PROGRAM Motion_Step_ST
VAR
    Vision_OK_Trig     : R_TRIG;             // 비전 OK 상승엣지(결과 캡처)
    VisionQueue        : FB_VisionDataQueue; // 비전 결과 큐(덮어쓰기 방지, 용량5)
    Vis_Item           : ST_VisionData;      // 큐 push 용 스크래치
    Vis_Head           : ST_VisionData;      // 큐 pop(Head) 용 스크래치
    Cam_Trig_Pos_Buf   : LREAL;              // 소비된 부품의 캠트리거 위치(Target X 보정 기준)
    Active_ID          : DINT;               // 현재 처리(압입) 중 부품의 비전 인식 ID
    Skip_Event         : BOOL;               // 이번 스캔 프레스 실패(skip) 발생 — NG 부저 트리거(매 스캔 클리어)
    NG_Playing         : BOOL;               // NG 모스 부저 재생 중
    NG_Timer           : TON;                // NG 패턴 경과시간 타이머(한 번 ≈ 1초)
    Cand_Target_X      : LREAL;              // pop 후보 부품의 현재 Target X (도달성 판단)
    Data_Initial       : BOOL;               // 캡처 직후 Data_Read/Vision_OK 초기화 예약
    Vision_Copy_Status : BOOL;               // 비전 캡처 게이트(오토 전용: Auto AND Safety)
    Stop_Req           : BOOL;               // (옵션) 프레스 실패 정지 요청 래치 — No=0(안전·X기어해제)에서 All_Motor_Stop 적용
    Auto_Resume_Trig   : R_TRIG;             // 오토 재요청 상승엣지(정지 해제·복구)
    X_Coupled          : BOOL;               // X(Axis02) 기어 커플 상태 추적 — Press_Start에서 래치, Work_End_Position에서 해제
    Manual_Nudge       : BOOL;               // 림보(Auto·Manual 둘다 OFF) 탈출용 수동요청 넛지 플래그
    Z_Torque_Timer      : TON;               // 압입 토크 임계 도달 지속 확인(하강 가속 스파이크 오검출 방지)
    Z_Torque_Reach_Time : TIME := T#100MS;   // 토크 임계 도달 확정 지속시간 — 장비 튜닝
    Z_Stop_Timer        : TON;               // 토크완료 후 Z MC_Stop 정지 확인 디바운스
    Z_Stop_Conf_Vel     : LREAL := 1.0;      // 정지 판정 속도(이 미만이면 정지 완료) — 장비 튜닝
    Z_Stop_Conf_Time    : TIME := T#50MS;    // 정지 확정 지속시간
END_VAR

// 엣지 검출 (매 스캔)
Vision_OK_Trig(CLK := GVL_Vision.Vision_OK);

// 코일 초기화
GVL_Motion_Step.Motion_Start := FALSE;
GVL_Motion_Step.Target_Pos_Moving := FALSE;
GVL_Motion_Step.Axis02_Work_Wait := FALSE;
GVL_Motion_Step.Press_Start := FALSE;
GVL_Motion_Step.Z_Press_Start := FALSE;
GVL_Motion_Step.Axis04_Wait_Pos_Moving := FALSE;
GVL_Motion_Step.Axis02_Stop := FALSE;
GVL_Motion_Step.All_Axis_Wait_Pos_Moving := FALSE;
GVL_Motion_Step.Work_Comp_Target_Pos_Moving := FALSE;
GVL_Motion_Step.All_Initial := FALSE;
Skip_Event := FALSE;   // 매 스캔 클리어 (skip 발생 스캔만 TRUE)

// ===== 비전 결과 캡처 (덮어쓰기 방지) =====
// 모션 가능여부와 무관하게, 가깝게 들어온 Vision_OK 결과를 매 엣지마다 큐에 전부 적재.
IF GVL_System.Auto_Mode AND Vision_OK_Trig.Q THEN
    Vis_Item.ID                := GVL_Vision.Data_Read_ID;        // 인식 ID 스냅샷
    Vis_Item.X                 := GVL_Vision.Data_Read_X;
    Vis_Item.Y                 := GVL_Vision.Data_Read_Y;
    Vis_Item.Rot               := GVL_Vision.Data_Read_R;
    Vis_Item.Cam_Trig_Position := GVL_Vision.Cam_Trig_Position;   // 캡처 시점 캠트리거 위치 스냅샷
    IF VisionQueue.Push(Vis_Item) THEN
        GVL_Vision.Vision_Q_Overflow := FALSE;
    ELSE
        GVL_Vision.Vision_Q_Overflow := TRUE;   // 큐 만재 → 무음 유실 방지 경보(용량↑ 또는 프레스 처리율↑)
        // 큐 만재로 미적재 → skip 보고 (reason 3)
        GVL_Vision.Skipped_ID_Buf[GVL_Vision.Skip_Count MOD 256]     := Vis_Item.ID;
        GVL_Vision.Skipped_Reason_Buf[GVL_Vision.Skip_Count MOD 256] := 3;
        GVL_Vision.Skip_Count := GVL_Vision.Skip_Count + 1;
        Skip_Event := TRUE;   // 프레스 실패 → 부저 펄스 트리거
    END_IF
    Data_Initial := TRUE;   // Data_Read/Vision_OK 초기화 → 다음 결과 수신 준비
END_IF

GVL_Vision.Vision_Q_Count := VisionQueue.Count;   // HMI 모니터

// ===== 비전 큐 flush (pop 보호: stale 항목 영구잔류 방지) =====
// 오토 이탈 / 시스템 초기화 시 큐 비움. (사이클말 No=40 에서는 비우지 않음 — 대기 부품 보존)
IF NOT GVL_System.Auto_Mode OR GVL_System.All_Initial THEN
    VisionQueue.Clear();
    GVL_Vision.Vision_Q_Overflow := FALSE;
END_IF

// ===== 모션 시퀀스 (CASE: 스캔당 1스텝만 — 같은 스캔 cascade/stale 판정 방지) =====
IF GVL_System.Auto_Mode THEN

    // Target X 위치 계산 (스텝이 읽기 전, No<>0 일 때 매 스캔 갱신)
    IF GVL_Motion_Step.No <> 0 THEN
        GVL_Vision.Target_X_Real_Position_Data := GVL_Vision.Data_Buffer_X - (GVL_Encoder.Real_Position - Cam_Trig_Pos_Buf);
    END_IF

    CASE GVL_Motion_Step.No OF

        0:  // 큐에서 다음 부품 pop. Wait 위치를 지나친(도달불가) 부품은 폐기(실패), 도달 가능한 것만 적재.
            IF Stop_Req THEN
                // (옵션) 실패 정지 요청 대기 — 사이클 안전종료·X 기어해제 유휴에서만 정지 적용. pop 보류.
                GVL_System.All_Motor_Stop := TRUE;     // Auto 차단(→ 수동, 아래 넛지가 Manual 진입)
                GVL_Conv.Motor_STOP := TRUE;           // 실제 컨베이어 정지(Conv.TcPOU 가 모든 컨베이어 출력 OFF)
            ELSIF VisionQueue.Count > 0 THEN
                Vis_Head := VisionQueue.HeadData;    // 가장 오래된 항목
                Cand_Target_X := Vis_Head.X - (GVL_Encoder.Real_Position - Vis_Head.Cam_Trig_Position);
                IF Cand_Target_X >= GVL_Axis02.Wait_Position_Data THEN
                    // 아직 Wait 전 → 도달 가능 → 적재 + 시작
                    VisionQueue.Pop();
                    GVL_Vision.Data_Buffer_X := Vis_Head.X;
                    GVL_Vision.Data_Buffer_Y := Vis_Head.Y;
                    GVL_Vision.Data_Buffer_R := Vis_Head.Rot;
                    Cam_Trig_Pos_Buf         := Vis_Head.Cam_Trig_Position;
                    Active_ID                := Vis_Head.ID;     // 처리 중 부품 ID 보관(압입 시 보고)
                    GVL_Motion_Step.Motion_Start := TRUE; // not use
                    GVL_Motion_Step.No := 1;
                ELSE
                    // Wait 통과(이미 지나침, 도달불가) → 폐기 + skip 보고 (reason 1)
                    GVL_Vision.Skipped_ID_Buf[GVL_Vision.Skip_Count MOD 256]     := Vis_Head.ID;
                    GVL_Vision.Skipped_Reason_Buf[GVL_Vision.Skip_Count MOD 256] := 1;
                    GVL_Vision.Skip_Count := GVL_Vision.Skip_Count + 1;
                    Skip_Event := TRUE;   // 프레스 실패 → 부저 펄스 트리거
                    VisionQueue.Pop();   // 폐기, 다음 부품 시도
                END_IF
            END_IF

        1:  // R/Y 타겟 이동 시작 (블로킹 안 함 — 대기/sync 구간 병렬 이동, Z 프레스 직전 도달 확인)
            GVL_Motion_Step.Target_Pos_Moving := TRUE; // reference axis03_auto, axis01_auto
            GVL_Motion_Step.No := 5;

        5:  // Axis02 Work Wait (R/Y 병렬 이동 지속)
            GVL_Motion_Step.Target_Pos_Moving := TRUE;   // R/Y 계속 타겟으로
            GVL_Motion_Step.Axis02_Work_Wait := TRUE;
            IF GVL_Vision.Target_X_Real_Position_Data <= GVL_Axis02.Wait_Position_Data THEN
                GVL_Motion_Step.No := 10;
            END_IF

        10: // Press Start (sync). R/Y 타겟 도달 후에만 Z 프레스. R/Y 지연으로 압입범위 지나치면 실패 복귀.
            GVL_Motion_Step.Target_Pos_Moving := TRUE;   // R/Y 타겟 유지(sync 구간 병렬 이동)
            GVL_Motion_Step.Press_Start := TRUE;
            IF GVL_Vision.Target_X_Real_Position_Data <= (GVL_Axis02.Wait_Position_Data - GVL_Axis02.Sync_Data)
               AND GVL_Axis03.Target_Position AND GVL_Axis01.Target_Position THEN
                GVL_Motion_Step.Z_Press_Start := TRUE;
            END_IF

            // ===== 토크 압입 완료 판정 =====
            // 실제토크(GVL_Axis04.Torque_Actual, PDO)가 임계값(Press_Torque_Reach_Data) 이상으로
            // Z_Torque_Reach_Time 지속되면(가속 스파이크 오검출 방지) 목표 위치 미도달이어도 토크한계 도달로 완료.
            Z_Torque_Timer(IN := GVL_Motion_Step.Z_Press_Start
                                 AND ABS(GVL_Axis04.Torque_Actual) >= GVL_Axis04.Press_Torque_Reach_Data
                                 AND NOT GVL_Axis04.Work_End_Position,
                           PT := Z_Torque_Reach_Time);

            IF GVL_Axis04.Work_End_Position THEN
                // 정상(위치도달) 완료 — 기존 경로. 무손실 압입 ID 보고: 현재 count 슬롯에 ID 기록 → count 증가
                GVL_Vision.Pressed_ID_Buf[GVL_Vision.Press_Count MOD 256] := Active_ID;
                GVL_Vision.Press_Count := GVL_Vision.Press_Count + 1;   // vision은 Press_Count 증가분만큼 Buf 읽음
                GVL_Motion_Step.No := 20;
            ELSIF Z_Torque_Timer.Q THEN
                // 토크한계 도달 완료 — 위치 미도달(눌러박힘)이라 press MoveAbsolute 를 MC_Stop 으로 끊어야 함(No=15).
                // 컨베이어/부품 눌러박힘으로 Work_End_Position 이 안 떠 No=10 에 머물며 계속 누르던 hang 방지.
                GVL_Vision.Pressed_ID_Buf[GVL_Vision.Press_Count MOD 256] := Active_ID;
                GVL_Vision.Press_Count := GVL_Vision.Press_Count + 1;
                GVL_Motion_Step.No := 15;
            ELSIF GVL_Vision.Target_X_Real_Position_Data < 0
                  AND NOT GVL_Motion_Step.Z_Press_Start THEN
                // 미압입(R/Y 지연) abort → skip 보고 (reason 2)
                GVL_Vision.Skipped_ID_Buf[GVL_Vision.Skip_Count MOD 256]     := Active_ID;
                GVL_Vision.Skipped_Reason_Buf[GVL_Vision.Skip_Count MOD 256] := 2;
                GVL_Vision.Skip_Count := GVL_Vision.Skip_Count + 1;
                Skip_Event := TRUE;   // 프레스 실패 → 부저 펄스 트리거
                GVL_Motion_Step.No := 25;   // Z 미진입, 부품이 0(센서 닿기 전 한계) 지나침 → No=25 MC_Stop 복귀
            END_IF

        15: // 토크 압입 완료 후 Z 강제정지(MC_Stop) → 정지 확인 → 복귀(No=20)
            // press MoveAbsolute 는 Execute 를 떨궈도 안 멈추므로(계속 목표로 누름) Z MC_Stop(Axis04_Stop_01)로 확실히 끊는다.
            // GVL_Main_Step.Press_Stop → Axis04_Status 의 MC_Stop Execute(전용 훅). 정지 확인 후 해제해야 다음 복귀 move 가능.
            Z_Stop_Timer(IN := ABS(GVL_Axis04.Real_Velocity) < Z_Stop_Conf_Vel, PT := Z_Stop_Conf_Time);
            IF Z_Stop_Timer.Q THEN
                GVL_Main_Step.Press_Stop := FALSE;   // MC_Stop 해제 → No=20 Wait 복귀 move 실행 가능
                GVL_Motion_Step.No := 20;
            ELSE
                GVL_Main_Step.Press_Stop := TRUE;    // Z MC_Stop 유지(press 정지)
            END_IF

        20: // Axis04 Wait Pos Moving
            IF GVL_Axis02.Real_Position <-1 THEN
                GVL_Motion_Step.Press_Start := FALSE;
                GVL_Motion_Step.Axis04_Wait_Pos_Moving := TRUE;
                GVL_Motion_Step.No := 25;
            END_IF
            IF GVL_Axis02.Real_Position <= (GVL_Axis02.Work_End_Position_Data + 10) THEN
                GVL_Motion_Step.Axis04_Wait_Pos_Moving := TRUE;
            END_IF
            IF GVL_Axis02.Real_Position <= GVL_Axis02.Work_End_Position_Data THEN
                GVL_Motion_Step.No := 25;
            END_IF

        25: // Axis02 Stop
            GVL_Motion_Step.Axis02_Stop := TRUE;
            IF GVL_Axis02.Work_End_Position THEN
                GVL_Motion_Step.No := 30;
            END_IF

        30: // All Axis Wait Pos Moving
            GVL_Motion_Step.All_Axis_Wait_Pos_Moving := TRUE;
            IF GVL_System.ALL_Wait_Position THEN
                GVL_Motion_Step.No := 40;
            END_IF

        40: // 사이클말 — All Initial + 버퍼/카피완료 초기화 (비전 큐는 비우지 않음: 대기 부품 보존)
            GVL_Motion_Step.All_Initial := TRUE;
            GVL_Vision.Data_Buffer_X := 0;
            GVL_Vision.Data_Buffer_Y := 0;
            GVL_Vision.Data_Buffer_R := 0;
            GVL_Vision.Target_X_Real_Position_Data := 0;
            GVL_Motion_Step.No := 0;

    ELSE
        GVL_Motion_Step.No := 0;   // 미정의 스텝값 → 안전 복귀(유휴)

    END_CASE

END_IF

// ===== X 기어 커플 추적 + Auto 이탈 시 강제 디커플 (수동전환·안전 등 어떤 이유로든 기어인 방치 방지) =====
// 기존엔 디커플 체인(Axis02_Stop→MC_Stop→MC_GearOut)이 Auto No=25 에서만 트리거 → Auto 빠지면 X 기어인 잔류.
// Press_Start(기어인)에서 커플 래치, Work_End_Position(MC_GearOut.Done)에서 해제.
IF GVL_Motion_Step.Press_Start THEN
    X_Coupled := TRUE;
END_IF
IF GVL_Axis02.Work_End_Position THEN
    X_Coupled := FALSE;
END_IF
// Auto 가 빠졌는데 X가 아직 커플이면 → No 머신과 무관하게 디커플 체인 강제 구동(Axis02_Command 는 매 스캔 실행).
// 디커플 완료 시 X_Coupled 해제 → 코일초기화로 Axis02_Stop 자동 release → 수동 조그 가능.
IF X_Coupled AND NOT GVL_System.Auto_Mode THEN
    GVL_Motion_Step.Axis02_Stop := TRUE;
END_IF

// ===== Z 정지훅(Press_Stop) 안전 해제 =====
// 토크완료 정지(No=15)용 Z MC_Stop 훅. 오토 이탈·초기화 시 래치 잔류로 Z가 정지에 물려 수동조작·복구를
// 방해하지 않도록 해제. (No=15 정상 진행 시엔 그 스텝에서 정지확인 후 스스로 해제)
IF NOT GVL_System.Auto_Mode OR GVL_System.All_Initial THEN
    GVL_Main_Step.Press_Stop := FALSE;
END_IF

// Vision 데이터 초기화 (캡처 직후 다음 결과 수신 준비) =====
IF Data_Initial OR GVL_System.All_Initial THEN
    GVL_Vision.Data_Read_X := 0;
    GVL_Vision.Data_Read_Y := 0;
    GVL_Vision.Data_Read_R := 0;
    GVL_Vision.Vision_OK := FALSE;
    Data_Initial := FALSE;
END_IF

// ===== 프레스 실패(비전 왔는데 미압입) 부저 — "NG" 모스부호 (N:―· G:――·), 알람부저와 구분 =====
// 단위 60ms, 한 번 재생 ≈ 1초. skip 시 1회 재생. 중지·에러 없이 부저만, System 부저에 OR(비파괴).
IF NG_Timer.Q THEN
    NG_Playing := FALSE;
END_IF
IF Skip_Event THEN
    NG_Playing := TRUE;   // 실패 → NG 재생 시작(재생 중 추가 실패는 현재 재생 끝난 뒤 새로 시작)
END_IF
NG_Timer(IN := NG_Playing, PT := T#1020MS);
GVL_System.Buzzer := GVL_System.Buzzer OR (NG_Playing AND (
       (NG_Timer.ET <  T#180MS)                                  // N: dash(―)
    OR (NG_Timer.ET >= T#240MS AND NG_Timer.ET < T#300MS)        // N: dot(·)
    OR (NG_Timer.ET >= T#480MS AND NG_Timer.ET < T#660MS)        // G: dash(―)
    OR (NG_Timer.ET >= T#720MS AND NG_Timer.ET < T#900MS)        // G: dash(―)
    OR (NG_Timer.ET >= T#960MS AND NG_Timer.ET < T#1020MS)));    // G: dot(·)

// ===== (옵션) 프레스 실패 시 컨베이어 정지 + 수동 전환 — vision 이 GVL_Vision.Stop_On_Fail 로 ON/OFF =====
// 실패(skip) → Stop_Req 래치. 실제 정지는 No=0(사이클 안전종료·X 기어해제)에서 All_Motor_Stop 적용(위 CASE 0).
// All_Motor_Stop=TRUE → Auto 차단(→ 수동, 넛지가 Manual 진입) / Motor_STOP=TRUE → 컨베이어 정지(Conv.TcPOU). 알람/에러 없음. 수동 조작은 안 막음.
// 복구: 오토 재요청(HMI_Auto_Mode) 상승엣지 또는 리셋(All_Initial) 시 Stop_Req·All_Motor_Stop·Motor_STOP 해제.
IF Skip_Event AND GVL_Vision.Stop_On_Fail THEN
    Stop_Req := TRUE;
END_IF
Auto_Resume_Trig(CLK := GVL_System.HMI_Auto_Mode);
IF Auto_Resume_Trig.Q OR GVL_System.All_Initial THEN
    Stop_Req := FALSE;
    GVL_System.All_Motor_Stop := FALSE;
    GVL_Conv.Motor_STOP := FALSE;
END_IF

// ===== 림보(Auto·Manual 둘 다 OFF) 자동 탈출 → 수동 진입 =====
// Manual_Mode 진입은 (HMI_Manual_Mode AND NOT Each_Motor_Busy) 게이트라, 동작 중(gear-in/압입) 모드전환 시
// Auto 자기유지만 끊겨 Auto OFF·Manual 못 들어가는 림보 발생(모멘터리 수동버튼·fail-stop 공통).
// 모터 정지·안전·오토요청 아님이면 수동요청을 넣어 Manual 을 래치시키고, 진입되면 떼어냄.
// (HMI 는 버튼 누를 때만 HMI_Manual_Mode 를 쓰므로 평소엔 건드리지 않아 충돌 없음)
IF NOT GVL_System.Auto_Mode AND NOT GVL_System.Manual_Mode
   AND GVL_System.Safety_ALL_OK AND NOT GVL_System.Each_Motor_Busy
   AND NOT GVL_System.HMI_Auto_Mode THEN
    GVL_System.HMI_Manual_Mode := TRUE;    // 수동 진입 넛지
    Manual_Nudge := TRUE;
ELSIF Manual_Nudge THEN
    GVL_System.HMI_Manual_Mode := FALSE;   // 넛지로 set 한 것만 해제(진입 완료 후) — 오토 복귀 막지 않게
    Manual_Nudge := FALSE;
END_IF

END_PROGRAM

(* stored: Version 1.1.0.1, ProductVersion 3.1.4024.16
   POU Motion_Step_ST: Id {ac3913c8-2e13-4a7b-9725-7ff41cb7600e}, SpecialFunc None *)
